Staubli VAL3: Main_app.pjx

--- Main_app.pjx ---
Parameters version=s8.15.3Cs9_BS3337 stackSize=200000 millimeterUnit=true
Program file=AlterCtrl.pgx
Program file=DismountBolt.pgx
Program file=DismountGripper.pgx
Program file=ForceSensor.pgx
Program file=Init.pgx
Program file=IO.pgx
Program file=ManualJoint.pgx
Program file=MountBolt.pgx
Program file=MountGripper.pgx
Program file=MovementCtrl.pgx
Program file=OpcInterface.pgx
Program file=start.pgx
Program file=stop.pgx
Program file=ToolChanger.pgx
Data file=Main_app.dtx
Library alias=Test path=Disk://Test1/Test1.pjx
Library alias=Su path=Disk://safeUtilities/safeUtilities.pjx

--- Main_app.dtx ---
bool bBooltoNum
bool bBtnCtrlOpc
bool bBtnIntercambio
bool bError
public bool bEstAtornillador = true
public bool bEstPinza = true
public bool bHerramientaRobot = true
bool bOk
public bool bTLocked
public bool bTUnlocked = true
public bool btnToolChangeBolt
public bool btnToolChangeGrip
bool validPos
dio dChangerValve = {link=ValveIO\valve1}
dio dDioEstAtornillador = {link=CE061C2D-63EF-47EF-A59E-9D0AF6F8F85C}
dio dDioEstPinza = {link=09F12A79-E04E-419B-9AAF-7725DDDBD1AC}
dio dDioHerramientaRobot = {link=7E390559-96A8-403A-B445-689BBF355DEA}
dio dDioTLocked = {link=F2CD6568-BB9E-49C8-A7B4-91D8A66F9C51}
dio dDioTUnlocked = {link=60862B78-E473-4D73-B0A1-35126C8FEF27}
frame fHaption = {x=107.807516, y=-386.531428, z=887.560715, rx=-89.0477411, ry=-149.698587, rz=0.421407, fatherId=world[0]}
frame fToolChange = {x=615.030242, y=458.213417, z=150.671162, rx=-90.0936151, ry=30.458364, rz=89.118179, fatherId=world[0]}
jointRx jChange = {j1=-4.0714236, j2=-3.552111, j3=129.273225, j4=106.087665, j5=68.799532, j6=6.346847}
jointRx jHome = {j1=57.800006, j2=-37.780028, j3=119.215944, j4=179.0580443, j5=81.384924, j6=-131.0356711}
public jointRx jInitial = {j1=57.800006, j2=-37.780028, j3=119.215944, j4=179.0580443, j5=81.384924, j6=-131.0356711}
public jointRx jJointRx
jointRx jResult
jointRx jTouch = {j1=60.497505, j2=-107.87914, j3=120.00337332, j4=178.372552, j5=-48.125989, j6=4.636406}
mdesc mAppro = {accel=5, vel=5, decel=5, leave=1, reach=1}
mdesc mChange = {accel=10, vel=10, decel=10, leave=10, reach=10}
mdesc mNomSpeed = {accel=50, vel=50, decel=50}
public num OPCf1
public num OPCf2
public num OPCf3
public num OPCf4
public num OPCf5
public num OPCf6
public num OPCj1
public num OPCj2
public num OPCj3
public num OPCj4
public num OPCj5
public num OPCj6
public num OPCrx
public num OPCry
public num OPCrz
public num OPCx
public num OPCy
public num OPCz
num nCmd[6]
num nCmdTrans[6]
num nI
num nJ
public num nListForces[6]
num nPos
num nRawUdp[48]
num nState
num nTemp
public pointRx pActualPos
pointRx pPointRx
pointRx pTest = {x=-252.530153, y=263.294912, z=427.370916, rx=5.121571, ry=-7.129797, rz=162.640171}
pointRx pTool1 = {x=26.46, y=-161.846445, z=25.66398, rx=0.739769, ry=-0.0144029, rz=-134.866663, shoulder=lefty, elbow=epositive, wrist=wpositive, fatherId=fToolChange[0]}
pointRx pTool2 = {x=24.417771, y=213.35041, z=25.529958, rx=-0.30514, ry=-0.197907, rz=46.419643, shoulder=lefty, elbow=epositive, wrist=wpositive, fatherId=fToolChange[0]}
string sInfo = "Cogiendo el atornillador."
string sOutput = "No se ha podido dar potencia al brazo"
string sStringRaw[48]
tool tAtornillador = {x=-0.0903, y=-165.0894, z=43.1596, fatherId=tChanger[0]}
tool tChanger = {z=62.5, fatherId=flange[0], ioLink=ValveIO\valve1, ioOpen=0.5, ioClose=0.5}
tool tPinza = {y=48.1055, z=146.1642, fatherId=tChanger[0]}
tool tPuntero = {z=118, fatherId=flange[0]}
tool tTeach = {z=90, fatherId=flange[0]}
jointRx jGimbal = {j6=1}
public num nSpeedRate
public dio dDioMoveGripper = {link=B2194EAF-1145-4C79-9BA9-5960C08FF7FC}
public bool bMoveGripper
public bool bLockRotation
public bool bManualJoint
public bool bModeChanged
public num OPCj1cmd
public num OPCj2cmd
public num OPCj3cmd
public num OPCj4cmd
public num OPCj5cmd
public num OPCj6cmd
public bool bCogerPinza
public bool bCogerAtornillador
public bool bDejarPinza
public bool bDejarAtornillador
jointRx jStart = {j1=-6.36110936292703E-15, j2=4.98, j3=-90.18, j4=1.4230002260189E-21, j5=85.08, j6=6.36110860462371E-15}
bool bSupervisor
num countstring
num countrecord
bool flagactive
num lastReceived
dio dDioDoor1Status = {link=7E2C1981-2091-4168-A4C7-3B8F54F93892}
dio dDioDoor2Status = {link=DD4B0AAB-BB16-4B26-8EC1-F4B17697477E}
dio dDioEmergencyButton = {link=70CCD0F6-6BE7-4533-984C-B059D9950979}
dio dESbutton = {link=Rsi9IO\IusoA1}
dio dDoor1 = {link=Rsi9IO\IusiB1}
dio dDoor2 = {link=Rsi9IO\IusiA1}
num nStart
num nDelay
public dio diJ207J208_RE_PNS_I6 = {link=09F12A79-E04E-419B-9AAF-7725DDDBD1AC}
public dio doJ207J208_RE_PNS_Q6 = {link=5F8C0500-A0C2-418B-B33F-DA7D83872BF3}
public dio diJ207J208_RE_PNS_I2 = {link=60862B78-E473-4D73-B0A1-35126C8FEF27}
public dio doJ207J208_RE_PNS_Q5 = {link=70CCD0F6-6BE7-4533-984C-B059D9950979}
public dio doJ207J208_RE_PNS_Q3 = {link=7E2C1981-2091-4168-A4C7-3B8F54F93892}
public dio diJ207J208_RE_PNS_I1 = {link=7E390559-96A8-403A-B445-689BBF355DEA}
public dio diJ207J208_RE_PNS_I5 = {link=826855D7-B3BE-4D72-B5FB-E89AA8CE1BC8}
public dio doJ207J208_RE_PNS_Q7 = {link=89E313F4-BC69-4F53-99A0-AECEC5F380AE}
public dio doJ207J208_RE_PNS_Q2 = {link=8EED7CAF-566F-42FA-AB95-4CE736BA248A}
public dio doJ207J208_RE_PNS_Q1 = {link=957CEE52-2BF5-4DF0-8E67-FA620ACF6C14}
public dio doJ207J208_RE_PNS_Q0 = {link=B2194EAF-1145-4C79-9BA9-5960C08FF7FC}
public dio diJ207J208_RE_PNS_I7 = {link=CE061C2D-63EF-47EF-A59E-9D0AF6F8F85C}
public dio diJ207J208_RE_PNS_I4 = {link=D971BF12-E116-4771-AC73-77C32A945796}
public dio doJ207J208_RE_PNS_Q4 = {link=DD4B0AAB-BB16-4B26-8EC1-F4B17697477E}
public dio diJ207J208_RE_PNS_I3 = {link=ECDEAE6F-FADA-4468-909E-1E4B6F2B874F}
public dio diJ207J208_RE_PNS_I0 = {link=F2CD6568-BB9E-49C8-A7B4-91D8A66F9C51}
public sio SocketTCP = {link=Socket\ReceiveTcp}
public sio SocketUDP = {link=UdpSocket\ReceiveUdp}
num desordenados
num OpcPrecisionMovement
trsf trAlter
num nAlterBeginState
pointRx pFinishAlter = {x=-336.628720241718, y=50, z=505.159108540589, rx=-5.05493480877665E-23, ry=1.40872651758736E-05, rz=-1.15631870617668E-21, shoulder=righty, elbow=enegative, wrist=wpositive, fatherId=world[0]}
trsf trAlterMove
num OpcStepsMovement
num nAlterState
num nAlterEndState
pointRx pStart = {x=-336.829738845272, y=49.9999961803571, z=558.957317821961, rx=2.83367334814845E-09, ry=-0.115117715818688, rz=2.8115150816022E-12, shoulder=righty, elbow=enegative, wrist=wpositive, fatherId=world[0]}
num nRecordCmd[2010 3]
num nRecordCmdX[10000]
num nRecordCmdY[10000]
num nRecordCmdID[10000]
string sStringHistorical[10000]
bool almacenar
sio SocketUDPForceSensor = {link=UdpSocket\SocketUDPForceSensor}
num nRequestUDP[8]
num nrxforce
num nDiagSocket
num nDiagSocket2
num nResponseUDP[36]
num nResponses
num Fx
num Fy
num Fz
num Tx
num Ty
num Tz
num nTestfB[36]
num nTestfBIN[288]
num i
num bytenum
num cociente
num resto
num HEXNUMBER[4 2]
num DECNUMBER
num j
num FxLimit
num FyLimit
num FzLimit
num TxLimit
num TyLimit
num TzLimit
bool followHuman
bool bSupervisorForce
pointRx pPress1 = {x=-336.870168433842, y=49.999992370606, z=579.007588648422, rx=2.8335220482869E-09, ry=-0.115113873837275, rz=2.84048267905755E-12, shoulder=righty, elbow=enegative, wrist=wpositive, fatherId=world[0]}
pointRx pRelease1 = {x=-336.829643365744, y=-50.1476616059199, z=558.909800775024, rx=-9.93639403181191E-07, ry=-0.115115185933709, rz=-9.61953709022073E-07, shoulder=righty, elbow=enegative, wrist=wpositive, fatherId=world[0]}
pointRx pPress2 = {x=-336.870134367357, y=-50.1476774705417, z=578.993918901558, rx=-2.56189918387667E-06, ry=-0.115109572206669, rz=-2.47515326511544E-06, shoulder=righty, elbow=enegative, wrist=wpositive, fatherId=world[0]}
pointRx pRelease2 = {x=-336.829650546973, y=-150.228261555763, z=558.909800434958, rx=-1.72565131768918E-06, ry=-0.11511397198566, rz=-1.69662426766672E-06, shoulder=righty, elbow=enegative, wrist=wpositive, fatherId=world[0]}
pointRx pPress3 = {x=-336.86978960782, y=-150.228255444793, z=578.871206987795, rx=-3.03400370196542E-07, ry=-0.115116778365496, rz=-2.63029287251087E-06, shoulder=righty, elbow=enegative, wrist=wpositive, fatherId=world[0]}
string sOPCRobotyReady
bool OpcPreciseMode
pointRx pSlide1 = {x=197.7, y=-267.76, z=591.67, rz=17.74, fatherId=world[0]}
pointRx pSlide2 = {x=-197.7, y=-267.76, z=595.22, rz=17.74, fatherId=world[0]}
pointRx pSlide3 = {x=-269.92, y=-408.17, z=595.21, rz=17.74, fatherId=world[0]}
sio SocketUDPMySensor = {link=UdpSocket\SocketUDPMySensor}
public num FxFlag
public num FyFlag
public num FzFlag
num OPCrxcmdOut
num OPCrycmdOut
num OPCrzcmdOut
num OpcStepsRotation
bool OPCGoHoming
bool OpcPreciseModePrevious
num auxencod
num nReplyMySensor[24]
public bool OPCChangeTool
bool flagOnceChangeTool
bool flagAlter
bool launchAlter
bool launchManualJoint
bool launchToolChange
jointRx jHere
bool OPCSetZeroForces
bool prevlaunchAlter
bool prevlaunchManualJoint
bool prevlaunchToolChange
jointRx jResumeAlter = {j2=4.98, j3=-90.18, j5=85.08}

--- start.pgx ---
program start()
begin

  bLockRotation = true
  //call Su:startupCheck(false,true,true,nState)
  sOPCRobotyReady = "Connected"

  if true
    //EVS volver a activar este if
    if true
      enablePower()
      if(watch(isPowered(),5)==false)
        sOutput="No se ha podido dar potencia al brazo"
        popUpMsg(sOutput,3)
      endIf
      setMonitorSpeed(100)
      bError=false
      taskCreate "Init",20,Init()
      taskCreate "IOread",20,IO()
      //EN ESTA TAREA SE LE DA POTENCIA AL BRAZO
      //taskCreate "ToolChange",50,ToolChanger()
      //taskCreate "PressTest", 50 , ForceTest()
      taskCreate "PositionCtrl",100,MovementCtrl()
      //taskCreateSync "HmiOpcUA",0.01,bSupervisor ,OpcInterface()
      taskCreate "HmiOpcUA",100,OpcInterface()
      taskCreateSync "ForceSensor",0.002,bSupervisorForce,ForceSensor()

    endIf

  endIf

end

--- AlterCtrl.pgx ---
program AlterCtrl()
begin

  for nPos=0 to 47 step 1
    nRawUdp[nPos] = 0
    endFor

    clearBuffer(SocketUDP)
    //
    // Waits until an moveAlter is being execute.
    do
      nAlterBeginState=alterBegin(tChanger,mNomSpeed)
      alterMovel(pFinishAlter,tChanger,mNomSpeed)
    until nAlterBeginState==1
    //This string is changed in OPCInterface
    sOPCRobotyReady = "Connected"

    //Recalculate Alter's trsf until finish moveAlter
    while nAlterBeginState==1

      sioGet(SocketUDP,nRawUdp)


      //Reset vector for translation
      for nPos=0 to 5 step 1
        nCmd[nPos]=0
      endFor

      //CONVERT RAW ASCII TO STRING
      for nPos=0 to 47 step 1
        sStringRaw[nPos]=chr(nRawUdp[nPos])
      endFor

      //CONVERT STRING TO 6 VELOCITY VALUES
      for nPos=0 to 5 step 1
        nI=8*nPos
        toNum(sStringRaw[nI+1],nTemp,bBooltoNum)
        nCmd[nPos]=nCmd[nPos]+nTemp*100
        toNum(sStringRaw[nI+2],nTemp,bBooltoNum)
        nCmd[nPos]=nCmd[nPos]+nTemp*10
        toNum(sStringRaw[nI+3],nTemp,bBooltoNum)
        nCmd[nPos]=nCmd[nPos]+nTemp
        toNum(sStringRaw[nI+5],nTemp,bBooltoNum)
        nCmd[nPos]=nCmd[nPos]+nTemp/10
        toNum(sStringRaw[nI+6],nTemp,bBooltoNum)
        nCmd[nPos]=nCmd[nPos]+nTemp/100

        //sStringRaw empieza con el signo del valor
        //Minus sign is 45 in ASCII
        if sStringRaw[nI+0]=="-"
          nCmd[nPos]=nCmd[nPos]*(-1)
        endIf
      endFor

      //Transformacion de angulos y escalado de velocidad
      nCmdTrans[0]=nCmd[0]*nSpeedRate/100
      nCmdTrans[1]=nCmd[1]*nSpeedRate/100
      nCmdTrans[2]=-nCmd[2]*nSpeedRate/100

      if nCmd[5] != lastReceived
        nRecordCmdX[countrecord] = OPCx
        nRecordCmdY[countrecord] = OPCy
        nRecordCmdID[countrecord] = nCmd[5]
        //nRecordCmd[countrecord, 1] = OPCy
        //nRecordCmd[countrecord, 2] = OPCz
        if nCmd[5] != lastReceived + 1
          desordenados = desordenados +1
          almacenar = true
        endIf
        for nPos=0 to 47 step 1
          sStringHistorical[countrecord] = insert (sStringHistorical[countrecord], sStringRaw[nPos], nPos)
        endFor
        countrecord = countrecord + 1
        lastReceived = nCmd[5]
        //logMsg(sStringRaw[nPos],4)
      endIf

      trAlterMove.x=nCmd[0]
      trAlterMove.y=nCmd[1]
      trAlterMove.z=nCmd[2]
      //Rotaciones se reciben por OPC en lugar del socket UDP
      trAlterMove.rx=OPCrxcmdOut
      trAlterMove.ry=OPCrycmdOut
      trAlterMove.rz=OPCrzcmdOut

      //Change movement ratio between robot and touch
      if OpcPreciseMode != OpcPreciseModePrevious
        if OpcPreciseMode
          OpcPrecisionMovement = 0.01
          OpcStepsMovement = 0.01
          OpcPreciseModePrevious = true
        else
          OpcPrecisionMovement = 0.1
          OpcStepsMovement = 0.1
          OpcPreciseModePrevious = false
        endIf
      endIf


      //MODO CONTROL POR POSICION-----------------------------------------------------------------------------------------------------
      if followHuman == false
        //EVS hay que filtrar para que no se mueva mas de una unidad la transformada cada 4ms (puede ser positivo o negativo)
        //trAlter permite definir desplazamiento respecto al ptB (o el que se haya usado en la ultima orden altermove
        //X
        //Desplazamiento +x
        if((trAlterMove.x-trAlter.x)>OpcPrecisionMovement) and (FxFlag != -1)
          trAlter.x=trAlter.x+OpcStepsMovement
          //Desplazamiento -x
        elseIf((trAlterMove.x-trAlter.x)<-OpcPrecisionMovement) and (FxFlag != 1)
          trAlter.x=trAlter.x-OpcStepsMovement
        endIf
        //Y
        //Desplazamiento +y
        if((trAlterMove.y-trAlter.y)>OpcPrecisionMovement) and (FyFlag != -1)
          trAlter.y=trAlter.y+OpcStepsMovement
          //Desplazamiento -y
        elseIf((trAlterMove.y-trAlter.y)<-OpcPrecisionMovement) and (FyFlag != 1)
          trAlter.y=trAlter.y-OpcStepsMovement
        endIf
        //Z
        //Desplazamiento +z
        if((trAlterMove.z-trAlter.z)>OpcPrecisionMovement) and (FzFlag != -1)
          trAlter.z=trAlter.z+OpcStepsMovement
          //Desplazamiento -z
        elseIf((trAlterMove.z-trAlter.z)<-OpcPrecisionMovement) and (FzFlag != 1)
          trAlter.z=trAlter.z-OpcStepsMovement
        endIf
        //rX
        if(trAlterMove.rx-trAlter.rx)>OpcPrecisionMovement
          trAlter.rx=trAlter.rx+OpcStepsRotation
        elseIf(trAlterMove.rx-trAlter.rx)<-OpcPrecisionMovement
          trAlter.rx=trAlter.rx-OpcStepsRotation
        endIf
        //rY
        if(trAlterMove.ry-trAlter.ry)>OpcPrecisionMovement
          trAlter.ry=trAlter.ry+OpcStepsRotation
        elseIf(trAlterMove.ry-trAlter.ry)<-OpcPrecisionMovement
          trAlter.ry=trAlter.ry-OpcStepsRotation
        endIf
        //rZ
        if(trAlterMove.rz-trAlter.rz)>OpcPrecisionMovement
          trAlter.rz=trAlter.rz+OpcStepsRotation
        elseIf(trAlterMove.rz-trAlter.rz)<-OpcPrecisionMovement
          trAlter.rz=trAlter.rz-OpcStepsRotation
        endIf

      else
        //MODO SEGUIMIENTO HUMANO ON----------------------------------------------------------------------------------------------------------

        //NECESITA FTSENSOR
        //Comprobar si la fuerza en el sentido de movimiento es mayor a la permitida
        if Fx > FxLimit
          trAlter.x = trAlter.x + OpcStepsMovement
        elseIf Fx < (-FxLimit)
          trAlter.x = trAlter.x - OpcStepsMovement
        endIf
        if Fy > FyLimit
          trAlter.y = trAlter.y + OpcStepsMovement
        elseIf Fy < (FyLimit*(-1))
          trAlter.y = trAlter.y - OpcStepsMovement
        endIf
        if Fz > FzLimit
          trAlter.z = trAlter.z + OpcStepsMovement
        elseIf Fz < (-FzLimit)
          trAlter.z = trAlter.z - OpcStepsMovement
        endIf


      endIf


      nAlterState=alter(trAlter)
      //sAlterState=toString("",nAlterState)+": "+sAlter[toString("",nAlterState)]

      pFinishAlter = here(tChanger,fToolChange)
      jResumeAlter = herej()
      delay(0)


    endWhile
    //
    nAlterEndState=alterEnd()
    //sAlterState=toString("",nAlterState)+": "+sAlterEnd[toString("",nAlterState)]
end

--- DismountBolt.pgx ---
program DismountBolt()
begin
  sInfo="Parking bolting tool..."
        movej(jChange,tChanger,mNomSpeed)

        bOk=watch(bTUnlocked==false and bTLocked==true,5)

        if bOk==true
          movej(appro(pTool2,{0,0,-200,0,0,0}),tChanger,mChange)
          waitEndMove()
          movel(pTool2,tChanger,mAppro)

          bOk=watch(bEstAtornillador==true,20)
          if bOk==true
            dChangerValve=true
            delay(0.1)
            bOk=watch(bTUnlocked==true and bTLocked==false,5)

            if bOk==true
              movel(appro(pTool2,{0,0,-100,0,0,0}),tChanger,mChange)
              bOk=watch(bHerramientaRobot==false,5)
              if bOk==true
                movej(jChange,tChanger,mNomSpeed)
                waitEndMove()

              else
                disablePower()
                userPageAlert("Error. Check parking station.")
                bError=true

              endIf

            else
              disablePower()
              userPageAlert("Error. Tool can not be unlocked, check neumatic circuit.")
              bError=true

            endIf

          else
            disablePower()
            userPageAlert("Error. Tool not detected at parking station")
            bError=true

          endIf

        else
          disablePower()
          userPageAlert("Error. Tool can not be unlocked, check neumatic circuit")
          bError=true
        endIf
end

--- DismountGripper.pgx ---
program DismountGripper()
begin
  sInfo="Parking gripper..."
        movej(jChange,tChanger,mNomSpeed)

        bOk=watch(bTUnlocked==false and bTLocked==true,5)

        if bOk==true
          movej(appro(pTool1,{0,0,-200,0,0,0}),tChanger,mChange)
          waitEndMove()
          movel(pTool1,tChanger,mAppro)

          bOk=watch(bEstPinza==true,20)
          if bOk==true
            dChangerValve=true
            delay(0.1)
            bOk=watch(bTUnlocked==true and bTLocked==false,30)
            //5
            if bOk==true
              movel(appro(pTool1,{0,0,-100,0,0,0}),tChanger,mChange)
              bOk=watch(bHerramientaRobot==false,5)
              if bOk==true
                movej(jChange,tChanger,mNomSpeed)
                waitEndMove()

              else
                disablePower()
                userPageAlert("Error. Check parking station.")
                bError=true

              endIf

            else
              disablePower()
              userPageAlert("Error. Tool can not be unlocked, check neumatic circuit.")
              bError=true

            endIf

          else
            disablePower()
            userPageAlert("Error. Tool not detected at parking station")
            bError=true

          endIf

        else
          disablePower()
          userPageAlert("Error. Tool can not be unlocked, check neumatic circuit")
          bError=true

        endIf
end

--- ForceSensor.pgx ---
program ForceSensor()
begin
  clearBuffer(SocketUDPForceSensor)
  clearBuffer(SocketUDPMySensor)
  while true

    //FRAME INIT = x1234  () COMMON TO ALL COMMANDS
    nRequestUDP[0] = 18
    nRequestUDP[1] = 52

    //COMMAND_SPEED	0x0082
    nRequestUDP[2] = 0
    nRequestUDP[3] = 130
    //DATA SPEED = 1
    nRequestUDP[4] = 0
    nRequestUDP[5] = 0
    nRequestUDP[6] = 0
    nRequestUDP[7] = 2
    sioSet(SocketUDPForceSensor,nRequestUDP,8)

    //COMMAND_FILTER	0x0081  /* Command for setting filter */ /* 0 = No filter; 1 = 500 Hz; 2 = 150 Hz; 3 = 50 Hz; 4 = 15 Hz; 5 = 5 Hz; 6 = 1.5 Hz */
    nRequestUDP[2] = 0
    nRequestUDP[3] = 129
    //FILTER = 1
    nRequestUDP[4] = 0
    nRequestUDP[5] = 0
    nRequestUDP[6] = 0
    nRequestUDP[7] = 1
    sioSet(SocketUDPForceSensor,nRequestUDP,8)

    //COMMAND_BIAS	0x0042  /* Command for toggle biasing */
    nRequestUDP[2] = 0
    nRequestUDP[3] = 66
    // BIASING_OFF		0x00    /* Biasing off */
    nRequestUDP[4] = 0
    nRequestUDP[5] = 0
    nRequestUDP[6] = 0
    nRequestUDP[7] = 1
    sioSet(SocketUDPForceSensor,nRequestUDP,8)

    //COMMAND_START	0x0002  /* Command for toggle biasing */
    nRequestUDP[2] = 0
    nRequestUDP[3] = 2
    // SAMPLE_COUNT = 10
    nRequestUDP[4] = 0
    nRequestUDP[5] = 0
    nRequestUDP[6] = 0
    nRequestUDP[7] = 0
    sioSet(SocketUDPForceSensor,nRequestUDP,8)

    //COMMAND_BIAS	0x0042  /* Command for toggle biasing */
    nRequestUDP[2] = 0
    nRequestUDP[3] = 66
    // BIASING_ON		0xFF    /* Biasing on */
    nRequestUDP[4] = 0
    nRequestUDP[5] = 0
    nRequestUDP[6] = 0
    nRequestUDP[7] = 255
    nDiagSocket2 = sioSet(SocketUDPForceSensor,nRequestUDP,8)
    nDiagSocket = sioGet(SocketUDPForceSensor,nResponseUDP)

    while nDiagSocket != -1
      nDiagSocket = sioGet(SocketUDPForceSensor,nResponseUDP)

//      for j = 0 to 11 step 1
//        nReplyMySensor[j] = nResponseUDP[j]
//      endFor

      //Decodificamos las 6 componentes F/T
      //Contador para las 6 componentes de F/T
      for j = 0 to 5 step 1
        //1 Conversion dec->hex
        //Contador para los 4 bytes de cada valor
        bytenum = 0

        while bytenum < 4
        nReplyMySensor[(4*j) + bytenum] = nResponseUDP[12 + (4*j) + bytenum ]
          cociente = nResponseUDP[12 + (4*j) + bytenum ]
          for i=0 to 1 step 1
            HEXNUMBER[bytenum,i] = cociente % 16
            cociente = roundDown(cociente / 16)
          endFor
          bytenum = bytenum + 1
        endWhile

        //2 Concatenar y convertir hex -> dec
        DECNUMBER = 0

        //Caso numero negativo (hacer previamente complemento a 1)
        if(HEXNUMBER[0,0] == 15)
          DECNUMBER = DECNUMBER + (15 - (HEXNUMBER[3,0]))*power(16, 0)
          DECNUMBER = DECNUMBER + (15 - (HEXNUMBER[3,1]))*power(16, 1)
          DECNUMBER = DECNUMBER + (15 - (HEXNUMBER[2,0]))*power(16, 2)
          DECNUMBER = DECNUMBER + (15 - (HEXNUMBER[2,1]))*power(16, 3)
          DECNUMBER = DECNUMBER + (15 - (HEXNUMBER[1,0]))*power(16, 4)
          DECNUMBER = DECNUMBER + (15 - (HEXNUMBER[1,1]))*power(16, 5)
          DECNUMBER = DECNUMBER + (15 - (HEXNUMBER[0,0]))*power(16, 6)
          DECNUMBER = DECNUMBER + (15 - (HEXNUMBER[0,1]))*power(16, 7)
          DECNUMBER = -DECNUMBER
          //Caso numero positivo
        else
          DECNUMBER = DECNUMBER + (HEXNUMBER[3,0])*power(16, 0)
          DECNUMBER = DECNUMBER + (HEXNUMBER[3,1])*power(16, 1)
          DECNUMBER = DECNUMBER + (HEXNUMBER[2,0])*power(16, 2)
          DECNUMBER = DECNUMBER + (HEXNUMBER[2,1])*power(16, 3)
          DECNUMBER = DECNUMBER + (HEXNUMBER[1,0])*power(16, 4)
          DECNUMBER = DECNUMBER + (HEXNUMBER[1,1])*power(16, 5)
          DECNUMBER = DECNUMBER + (HEXNUMBER[0,0])*power(16, 6)
          DECNUMBER = DECNUMBER + (HEXNUMBER[0,1])*power(16, 7)
          DECNUMBER = DECNUMBER
        endIf


        //Asignamos el resultado a cada valor F/T con su factor de escala
        auxencod = 0
        switch j
          case 0
            Fx =  DECNUMBER/10000
          break
          case 1
            Fy =  DECNUMBER/10000
          break
          case 2
            Fz =  DECNUMBER/10000
          break
          case 3
            Tx =  DECNUMBER/100000
          break
          case 4
            Ty =  DECNUMBER/100000
          break
          case 5
            Tz =  DECNUMBER/100000
          break

          default
          break
        endSwitch
      endFor

      //Comprobar si se superan los limites de fuerza en cada eje y activar flags para Unity
      if Fx > FxLimit
        FxFlag = 1
      elseIf Fx < (-FxLimit)
        FxFlag = -1
      else
        FxFlag = 0
      endIf

      if Fy > FyLimit
        FyFlag = 1
      elseIf Fy < (-FyLimit)
        FyFlag = -1
      else
        FyFlag = 0
      endIf

      if Fz > FzLimit
        FzFlag = 1
      elseIf Fz < (-FzLimit)
        FzFlag = -1
      else
        FzFlag = 0
      endIf



      //Datos enviados con payload adicional para experimentos de saturacion en la red
      sioSet(SocketUDPMySensor,nReplyMySensor,24)
      nResponses = nResponses + 1
      delay(0)
    endWhile

    //COMMAND_STOP	0x0000  /* Command for stop streaming */
    nRequestUDP[2] = 0
    nRequestUDP[3] = 0
    // BIASING_OFF		0x00    /* Biasing off */
    nRequestUDP[4] = 0
    nRequestUDP[5] = 0
    nRequestUDP[6] = 0
    nRequestUDP[7] = 0
    sioSet(SocketUDPForceSensor,nRequestUDP,8)
    delay(4)

  endWhile
end

--- Init.pgx ---
program Init()
begin

  clearBuffer(SocketUDP)
  resetMotion()

  launchAlter = true
  launchManualJoint = false
  launchToolChange = false

  OPCrxcmdOut = 0
  OPCrycmdOut = 0
  OPCrzcmdOut = 0
  FxLimit = 10
  FyLimit = 10
  FzLimit = 10
  OpcPrecisionMovement = 0.1
  OpcStepsRotation = 0.01
  OpcStepsMovement = 0.1
  OpcPreciseMode = false
  followHuman = false
  trAlterMove = {0,0,0,0,0,0}
  OPCGoHoming = false
  trAlter={0,0,0,0,0,0}
  delay(0)

end

--- IO.pgx ---
program IO()
begin

  //Read and process external controller information
  while bError==false

    nStart=clock()
    nDelay = clock()-nStart

    bEstAtornillador=dDioEstAtornillador
    bEstPinza=dDioEstPinza
    bHerramientaRobot=dDioHerramientaRobot
    bTLocked=dDioTLocked
    bTUnlocked=dDioTUnlocked
    dDioMoveGripper=bMoveGripper


    if dESbutton == true
      dDioEmergencyButton = true
    else
      dDioEmergencyButton = false
    endIf

    if dDoor1 == true
      dDioDoor1Status = true
    else
      dDioDoor1Status = false
    endIf

    if dDoor2 == true
      dDioDoor2Status = true
    else
      dDioDoor2Status = false
    endIf

    delay(0)
  endWhile

end

--- ManualJoint.pgx ---
program ManualJoint()
begin
  jHere = herej()
  OPCj1cmd = jHere.j1
  OPCj2cmd = jHere.j2
  OPCj3cmd = jHere.j3
  OPCj4cmd = jHere.j4
  OPCj5cmd = jHere.j5
  OPCj6cmd = jHere.j6

  while true
    jJointRx.j1=OPCj1cmd
    jJointRx.j2=OPCj2cmd
    jJointRx.j3=OPCj3cmd
    jJointRx.j4=OPCj4cmd
    jJointRx.j5=OPCj5cmd
    jJointRx.j6=OPCj6cmd
    movej(jJointRx,flange,mAppro)
    waitEndMove()
  endWhile
end

--- MountBolt.pgx ---
program MountBolt()
begin
  sInfo="Mounting bolting tool...."
        movej(jChange,tChanger,mNomSpeed)
        dChangerValve=true
        bOk=watch(bTUnlocked==true and bTLocked==false,5)

        if bOk==true
          movej(appro(pTool2,{0,0,-100,0,0,0}),tChanger,mChange)
          waitEndMove()
          movel(pTool2,tChanger,mAppro)
          bOk=watch(bHerramientaRobot==true,20)

          if bOk==true
            dChangerValve=false
            delay(0.1)
            bOk=watch(bTUnlocked==false and bTLocked==true,5)

            if bOk==true
              movel(appro(pTool2,{0,0,-200,0,0,0}),tChanger,mChange)
              movej(jChange,tChanger,mNomSpeed)
              waitEndMove()
              sInfo="Bolting tool ready"
            else
              disablePower()
              userPageAlert("Error. Tool not locked, check neumatic circuit.")
              bError=true

            endIf

          else
            disablePower()
            userPageAlert("Error. Tool can not be equiped., check position")
            bError=true

          endIf

        else
          disablePower()
          userPageAlert("Error. Tool can not be unlocked, check neumatic circuit.")
          bError=true

        endIf
end

--- MountGripper.pgx ---
program MountGripper()
  begin
  //1.-   CogerPinza()
        sInfo="Mounting griper...."
        movej(jChange,tChanger,mNomSpeed)
        dChangerValve=true
        bOk=watch(bTUnlocked==true and bTLocked==false,5)

        if bOk==true
          movej(appro(pTool1,{0,0,-100,0,0,0}),tChanger,mChange)
          waitEndMove()
          movel(pTool1,tChanger,mAppro)
          bOk=watch(bHerramientaRobot==true,20)

          if bOk==true
            dChangerValve=false
            delay(0.1)
            bOk=watch(bTUnlocked==false and bTLocked==true,5)

            if bOk==true
              movel(appro(pTool1,{0,0,-200,0,0,0}),tChanger,mChange)
              movej(jChange,tChanger,mNomSpeed)
              waitEndMove()
              sInfo="Griper ready"
            else
              disablePower()
              userPageAlert("Error. Tool not locked, check neumatic circuit.")
              bError=true

            endIf

          else
            disablePower()
            userPageAlert("Error. Tool can not be equiped., check position")
            bError=true

          endIf

        else
          disablePower()
          userPageAlert("Error. Tool can not be unlocked, check neumatic circuit.")
          bError=true

        endIf
        bCogerPinza=false

end

--- MovementCtrl.pgx ---
program MovementCtrl()
begin

  // Moves to start position.
  movej(jStart,flange,mNomSpeed)
  waitEndMove()



  while true
    //Detect if mode has been changed


    //Manage tasks if mode changed
    if launchAlter and launchAlter != prevlaunchAlter
      sOPCRobotyReady = "Restart"
      taskKill("ToolChange")
      taskKill("ManualCtrl")
      jResumeAlter.j3 = jResumeAlter.j3 + 1
      trAlter={0,0,0,0,0,0}
      movej(jResumeAlter,tChanger,mNomSpeed)
      waitEndMove()
      taskCreate "AlterCtrl",100,AlterCtrl()
      launchToolChange = false
      launchManualJoint = false
    endIf

    if launchManualJoint and launchManualJoint != prevlaunchManualJoint
      sOPCRobotyReady = "Restart"
      nAlterEndState=alterEnd()
      taskKill("ToolChange")
      taskKill("AlterCtrl")
      taskCreate "ManualCtrl",100,ManualJoint()
      launchToolChange = false
      launchAlter = false

    endIf

    if launchToolChange and launchToolChange != prevlaunchToolChange
      sOPCRobotyReady = "Restart"
      nAlterEndState=alterEnd()
      taskKill("AlterCtrl")
      taskKill("ManualCtrl")
      taskCreate "ToolChange",100,ToolChanger()
      launchAlter = false
      launchManualJoint = false
    endIf


//        if OPCGoHoming
//      while taskKill("PositionCtrl") != true
//        //ESPERAR A QUE LA TAREA SE CIERRE
//        delay(0)
//      endWhile
//      taskCreate "PositionCtrl",100,AlterCtrl()
//      taskCreate "Init",20,Init()
//    endIf

    prevlaunchAlter = launchAlter
    prevlaunchManualJoint = launchManualJoint
    prevlaunchToolChange = launchToolChange

    delay(0)
  endWhile
end

--- OpcInterface.pgx ---
program OpcInterface()
begin
  //Para poder escribir valores a través de OPC UA tienes que registrarte en el servidor con algun usuario (user:maintenance , pass: spec_cal)
  opcuaExport(sOPCRobotyReady,true)
  opcuaExport(OpcPreciseMode,true)
  opcuaExport(OpcPrecisionMovement,true)
  opcuaExport(OpcStepsMovement,true)
  opcuaExport(OpcStepsRotation,true)

  //opcuaExport(nRecordCmdX,true)
  //opcuaExport(nRecordCmdY,true)
  //opcuaExport(nRecordCmdID,true)
  opcuaExport(desordenados,true)
  opcuaExport(countrecord,true)

  opcuaExport(Fx,true)
  opcuaExport(Fy,true)
  opcuaExport(Fz,true)
  opcuaExport(Tx,true)
  opcuaExport(Ty,true)
  opcuaExport(Tz,true)
  opcuaExport(FxLimit,true)
  opcuaExport(FyLimit,true)
  opcuaExport(FzLimit,true)
  opcuaExport(TxLimit,true)
  opcuaExport(TyLimit,true)
  opcuaExport(TzLimit,true)
  opcuaExport(FxFlag,true)
  opcuaExport(FyFlag,true)
  opcuaExport(FzFlag,true)
  opcuaExport(followHuman,true)

  opcuaExport(OPCrxcmdOut,true)
  opcuaExport(OPCrycmdOut,true)
  opcuaExport(OPCrzcmdOut,true)
  opcuaExport(OPCGoHoming,true)
  opcuaExport(OPCChangeTool,true)

  opcuaExport(launchAlter,true)
  opcuaExport(launchManualJoint,true)
  opcuaExport(launchToolChange,true)
  opcuaExport(OPCSetZeroForces,true)
  opcuaExport(btnToolChangeBolt,true)
opcuaExport(btnToolChangeGrip,true)

  opcuaExport(OPCj1cmd,true)
  opcuaExport(OPCj2cmd,true)
  opcuaExport(OPCj3cmd,true)
  opcuaExport(OPCj4cmd,true)
  opcuaExport(OPCj5cmd,true)
  opcuaExport(OPCj6cmd,true)


  //Velocidad de inicio en el SCADA
  nSpeedRate=100



  while true

    //logMsg(toString("8.4", OPCx))


//    if OPCChangeTool
//      sOPCRobotyReady = "Restart"
//      if flagOnceChangeTool == false
//        while taskKill("PositionCtrl") != true
//          //ESPERAR A QUE LA TAREA SE CIERRE
//          delay(0)
//        endWhile
//        nAlterEndState=alterEnd()
//        resetMotion()
//        setMonitorSpeed(10)
//        movej(jChange,tChanger,mNomSpeed)
//        waitEndMove()
//        taskCreate "PositionCtrl",100,AlterCtrl()
//        //OPCChangeTool = false
//        flagOnceChangeTool = true
//      endIf
//    else
//      flagOnceChangeTool = false

//    endIf

    if OPCSetZeroForces
      taskKill("ForceSensor")
      taskCreateSync "ForceSensor",0.002,bSupervisorForce,ForceSensor()
      OPCSetZeroForces = false
    endIf

    delay(0)

  endWhile
end

--- ToolChanger.pgx ---
program ToolChanger()
begin


  //userPage("ToolChanger")
  //delay(0.5)
  //bOk=userPageConfirm("ATTENTION! Check the following points before press OK: 1-Tools are in place 2- Compressor and PLCs are powered 3-The arm can reach safely homing pose")
  //watch(bOk==true,120)

  bManualJoint = false
  btnToolChangeGrip = false
  btnToolChangeBolt = false
  bDejarPinza = false
  bDejarAtornillador = false


  //HABILITAMOS POTENCIA, HABILITAMOS FLAGS, PERO NO MANDAMOS MOVIMIENTOS DESDE ESTA TAREA
  if true
    enablePower()
    if(watch(isPowered(),5)==false)
      sOutput="Power is required, check the status."
      popUpMsg(sOutput,3)
    endIf

    // COMPROBAR QUE LAS HERRRAMIENTAS ESTAN EN LA ESTACION DE REPOSO O EQUIPADAS
    if bHerramientaRobot==true
      if bEstPinza==false and bEstAtornillador==false
        disablePower()
        userPageAlert("Error. Missing tool at parking station.")
        bError=true

      elseIf bEstPinza==true and bEstAtornillador==true
        disablePower()
        userPageAlert("Error. Tool sensors signal failure.")
        bError=true

      endIf
    endIf


    while bError==false

      delay(1)
      //CASOS EN LOS QUE NO HACEMOS NADA
      if btnToolChangeBolt==true and btnToolChangeGrip==true
        bCogerPinza=false
        bCogerAtornillador=false
        bDejarAtornillador=false
        bDejarPinza=false
        userPageAlert("Error. Two tools can not be equiped at the same time.")

        //HERRAMIENTAS EN REPOSO Y QUEREMOS EQUIPAR ALGO
      elseIf bHerramientaRobot==false and bEstAtornillador==true and bEstPinza==true and btnToolChangeGrip==true and btnToolChangeBolt==false
        //bCogerPinza=true
        call MountGripper()
      elseIf bHerramientaRobot==false and bEstAtornillador==true and bEstPinza==true and btnToolChangeBolt==true and btnToolChangeGrip==false
        //bCogerAtornillador=true
        call MountBolt()
        //HERRAMIENTA EQUIPADA Y QUEREMOS CAMBIAR A LA OTRA
      elseIf bHerramientaRobot==true and bEstAtornillador==true and bEstPinza==false and btnToolChangeBolt==true and btnToolChangeGrip==false
        //bDejarPinza=true
        call DismountGripper()
      elseIf bHerramientaRobot==true and bEstAtornillador==false and bEstPinza==true and btnToolChangeBolt==false and btnToolChangeGrip==true
        //bDejarAtornillador=true
        call DismountBolt()

        //HERRAMIENTA EQUIPADA Y QUEREMOS DEJARLA
      elseIf bHerramientaRobot==true and bEstAtornillador==true and bEstPinza==false and btnToolChangeBolt==false and btnToolChangeGrip==false
        //bDejarPinza=true
        call  DismountGripper()

      elseIf bHerramientaRobot==true and bEstAtornillador==false and bEstPinza==true and btnToolChangeBolt==false and btnToolChangeGrip==false
        //bDejarAtornillador=true
        call DismountBolt()

        //COMBINACIONES IMPOSIBLES
        //elseIf btnToolChangeBolt==false and btnToolChangeGrip==false
        //do nothing
        //        bCogerPinza=false
        //        bCogerAtornillador=false
        //        bDejarAtornillador=false
        //        bDejarPinza=false


      else
        //Exit while loop
        //       bCogerPinza=false
        //       bCogerAtornillador=false
        //     bDejarAtornillador=false
        //    bDejarPinza=false
        //     userPageAlert("Error. UNKNOWN COMBINATION......Tools are not in place or sensors are failing.")
        //   bError=true
      endIf

    endWhile

  else

    sInfo="Process has failed, check tool position and sensors."
    disablePower()

    delay(5)

  endIf

end
